FUNCTION_BLOCK FB_StateEStop IMPLEMENTS I_State
VAR
	_refMainStateMachine		: REFERENCE TO FB_MainStateMachine;
END_VAR

METHOD StopButtonPressed
END_METHOD

METHOD StartButtonPressed
END_METHOD

METHOD FB_init : BOOL
VAR_INPUT
	// if TRUE, the retain variables are initialized (warm start / cold start)
	bInitRetains			: BOOL;
	// if TRUE, the instance afterwards gets moved into the copy code (online
	// change)
	bInCopyCode				: BOOL;
	fbMainStateMachine		: REFERENCE TO FB_MainStateMachine;
END_VAR
_refMainStateMachine REF= fbMainStateMachine;
END_METHOD

METHOD SafetyAcknowledged
VAR_INPUT
END_VAR
_refMainStateMachine.SetState(_refMainStateMachine.ipStateInit);
END_METHOD

METHOD Execute
END_METHOD

METHOD SafetyTripped
VAR_INPUT
END_VAR
END_METHOD

END_FUNCTION_BLOCK

(* stored: Version 1.1.0.1, ProductVersion 3.1.4024.11
   POU FB_StateEStop: Id {f54b014d-f326-4723-be88-6f13db5d8daf}, SpecialFunc None
   Method StopButtonPressed: Id {0a1a9aca-495d-4051-b8f6-eebd2f604001}
   Method StartButtonPressed: Id {40b582c5-15c2-4625-9214-ceca93a65606}
   Method FB_init: Id {50d0ae89-8e9e-49ae-9389-acc70814cc80}
   Method SafetyAcknowledged: Id {5cddf761-b72b-4632-96c5-9e7ef79c977d}
   Method Execute: Id {9394d869-4e2b-4a71-a094-f42d5147ed92}
   Method SafetyTripped: Id {d9415e47-30ed-4951-a49c-b8be46bfc9d9} *)
